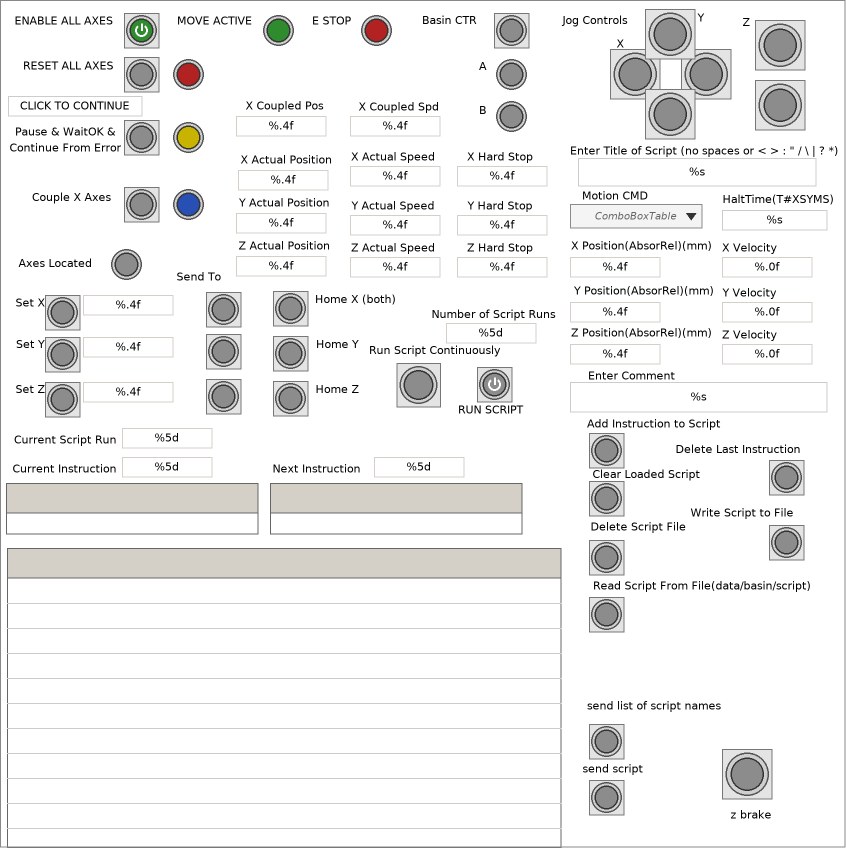
VISUALIZATION visMotorControl  // 846x848
    Label (12,58 113x16), "RESET ALL AXES"
    Label (12,126 107x12), "Pause & WaitOK &"
    Label (9,13 110x16), "ENABLE ALL AXES"
    Textfield (722,257 90x20), "%.0f", text variable: GVL_MOTION.InstructionBuffer.SetXVelocity
        OnMouseClick: write the text variable via InputWithLimits, min 1, max 300, title 'Enter Speed'
    Textfield (570,257 90x20), "%.4f", text variable: GVL_MOTION.InstructionBuffer.SetXPosition
        OnMouseClick: write the text variable via Default, min -200, max 1500
    Label (722,241 55x14), "X Velocity"
    Label (570,238 143x16), "X Position(AbsorRel)(mm)"
    Label (350,149 86x16), "X Actual Speed"
    Label (238,149 97x22), "X Actual Position"
    Textfield (350,166 90x20), "%.4f", text variable: GVL_MOTION.STATUS.xVelOut
    Textfield (238,170 90x20), "%.4f", text variable: GVL_MOTION.STATUS.xPosOut
    ComboBoxTable (570,204 132x24), variable: GVL_MOTION.InstructionBuffer.MotionCommand, data array: GVL_MOTION.xyzCMDSelect
        p1014161805: 4 - 0 + INT#1
        p3854506369: GVL_MOTION.xyzCMDSelect[INDEX]
    Label (564,185 102x22), "Motion CMD"
    PushSwitch (589,433 35x35), variable: GVL_MOTION.EXT_CTR.CMDADD, behaviour: TAP, style: Switch-PushSwitch-Gray
    Label (588,416 132x16), "Add Instruction to Script"
    PushSwitch (589,481 35x35), variable: GVL_MOTION.EXT_CTR.CMDCLR, behaviour: TOGGLE, style: Switch-PushSwitch-Gray
    Label (588,465 117x19), "Clear Loaded Script"
    Label (445,402 91x16), "RUN SCRIPT"
    PowerSwitch (477,367 35x35), variable: GVL_MOTION.EXT_CTR.CMDRUN, behaviour: TOGGLE, style: Switch-PowerSwitch-Gray
    Label (722,192 113x15), "HaltTime(T#XSYMS)"
    Textfield (722,210 105x20), "%s", text variable: GVL_MOTION.InstructionBuffer.pausetime
        OnMouseClick: write the text variable via Default, min 0, max 2000
    Label (554,12 82x17), "Jog Controls"
    PushSwitch (610,49 50x50), variable: GVL_MOTION.xJogBW, behaviour: TAP, style: Switch-PushSwitch-Gray
    PushSwitch (681,49 50x50), variable: GVL_MOTION.xJogFW, behaviour: TAP, style: Switch-PushSwitch-Gray
    Textfield (8,96 134x20), "CLICK TO CONTINUE", invisible if: GVL_MOTION.TxtBxWaitOK
    Lamp1 (171,57 35x35), variable: GVL_MOTION.STATUS.PowerError, style: Lamp-Lamp1-Red
    PushSwitch (45,295 35x35), variable: GVL_MOTION.EXT_CTR.SETXPOS, behaviour: TAP, style: Switch-PushSwitch-Gray
    PushSwitch (273,291 35x35), variable: GVL_MOTION.EXT_CTR.CMDHOMEX, behaviour: TAP, style: Switch-PushSwitch-Gray
    Label (14,295 33x16), "Set X"
    Label (313,291 85x17), "Home X (both)"
    Textfield (570,302 90x20), "%.4f", text variable: GVL_MOTION.InstructionBuffer.SetYPosition
        OnMouseClick: write the text variable via Default, min -200, max 1500
    Label (570,283 148x16), "Y Position(AbsorRel)(mm)"
    Textfield (722,302 90x20), "%.0f", text variable: GVL_MOTION.InstructionBuffer.SetYVelocity
        OnMouseClick: write the text variable via InputWithLimits, min 1, max 300, title 'Enter Speed'
    Label (722,286 55x14), "Y Velocity"
    Label (350,198 86x16), "Y Actual Speed"
    Label (236,192 97x22), "Y Actual Position"
    Textfield (350,215 90x20), "%.4f", text variable: GVL_MOTION.STATUS.yVelOut
    Textfield (236,213 90x20), "%.4f", text variable: GVL_MOTION.STATUS.yPosOut
    PushSwitch (45,337 35x35), variable: GVL_MOTION.EXT_CTR.SETYPOS, behaviour: TAP, style: Switch-PushSwitch-Gray
    Label (14,337 33x15), "Set Y"
    PushSwitch (645,9 50x50), variable: GVL_MOTION.yJogFW, behaviour: TAP, style: Switch-PushSwitch-Gray
    PushSwitch (645,89 50x50), variable: GVL_MOTION.yJogBW, behaviour: TAP, style: Switch-PushSwitch-Gray
    Label (6,141 119x14), "Continue From Error"
    Lamp1 (359,13 35x35), variable: GVL_MOTION.STATUS.eStop, style: Lamp-Lamp1-Red
    Label (300,13 63x16), "E STOP"
    PushSwitch (124,187 35x35), variable: GVL_MOTION.EXT_CTR.CMDCOUPLE, behaviour: TAP, style: Switch-PushSwitch-Gray
    Label (29,192 85x11), "Couple X Axes"
    Lamp1 (171,187 35x35), variable: GVL_MOTION.STATUS.xCoupled, style: Lamp-Lamp1-Blue
    Label (350,99 98x16), "X Coupled Spd"
    Label (236,95 97x22), "X Coupled Pos"
    Textfield (350,116 90x20), "%.4f", text variable: GVL_MOTION.xCOut.VelocityOut
    Textfield (236,116 90x20), "%.4f", text variable: GVL_MOTION.xCOut.PositionOut
    Label (693,9 16x18), "Y"
    Label (603,29 35x30), "X"
    PushSwitch (755,80 50x50), variable: GVL_MOTION.zJogBW, behaviour: TAP, style: Switch-PushSwitch-Gray
    PushSwitch (755,20 50x50), variable: GVL_MOTION.zJogFW, behaviour: TAP, style: Switch-PushSwitch-Gray
    Label (737,13 19x19), "Z"
    Label (350,240 86x16), "Z Actual Speed"
    Label (236,235 97x22), "Z Actual Position"
    Textfield (350,257 90x20), "%.4f", text variable: GVL_MOTION.STATUS.zVelOut
    Textfield (236,256 90x20), "%.4f", text variable: GVL_MOTION.STATUS.zPosOut
    Textfield (446,323 90x20), "%5d", text variable: GVL_MOTION.EXT_CTR.SCRIPTITERATIONS
        OnMouseClick: write the text variable via Default, min 1, title 'Enter Speed'
    Label (428,307 131x15), "Number of Script Runs"
    Label (12,255 87x17), "Axes Located"
    Table (6,483 252x51), data array: GVL_MOTION.Script[GVL_MOTION.CurInstruction]
        p3854506369: GVL_MOTION.Script[GVL_MOTION.CurInstruction].MotionCommand
        p1892666644: GVL_MOTION.Script[GVL_MOTION.CurInstruction].SetXPosition
        p338671338: GVL_MOTION.Script[GVL_MOTION.CurInstruction].SetXVelocity
        p2170511999: GVL_MOTION.Script[GVL_MOTION.CurInstruction].SetXAccel
        p3723444502: GVL_MOTION.Script[GVL_MOTION.CurInstruction].SetYPosition
        p1218418051: GVL_MOTION.Script[GVL_MOTION.CurInstruction].SetYVelocity
        p746581629: GVL_MOTION.Script[GVL_MOTION.CurInstruction].SetYAccel
        p3104783080: GVL_MOTION.Script[GVL_MOTION.CurInstruction].SetZPosition
        p2501879983: GVL_MOTION.Script[GVL_MOTION.CurInstruction].SetZVelocity
        p7306298: GVL_MOTION.Script[GVL_MOTION.CurInstruction].PauseTime
        p1933151965: GVL_MOTION.Script[GVL_MOTION.CurInstruction].Comment
        p511219082: xPos
        p1755163831: xVel
        p2237128397: yPos
        p505689113: yVel
        p4088588272: zPos
        p2243050616: zVel
    Label (368,343 134x15), "Run Script Continuously"
    PushSwitchLed (396,363 45x44), variable: GVL_MOTION.CMDLOOP_INT, behaviour: TOGGLE, style: Switch-PushSwitchLed-Gray
    Label (12,461 105x16), "Current Instruction"
    Textfield (122,457 90x20), "%5d", text variable: GVL_MOTION.CurInstruction
        OnMouseClick: write the text variable via Default
    Table (270,483 252x51), data array: GVL_MOTION.Script[GVL_MOTION.NextInstruction]
        p3854506369: GVL_MOTION.Script[GVL_MOTION.NextInstruction].MotionCommand
        p1892666644: GVL_MOTION.Script[GVL_MOTION.NextInstruction].SetXPosition
        p338671338: GVL_MOTION.Script[GVL_MOTION.NextInstruction].SetXVelocity
        p2170511999: GVL_MOTION.Script[GVL_MOTION.NextInstruction].SetXAccel
        p3723444502: GVL_MOTION.Script[GVL_MOTION.NextInstruction].SetYPosition
        p1218418051: GVL_MOTION.Script[GVL_MOTION.NextInstruction].SetYVelocity
        p746581629: GVL_MOTION.Script[GVL_MOTION.NextInstruction].SetYAccel
        p3104783080: GVL_MOTION.Script[GVL_MOTION.NextInstruction].SetZPosition
        p2501879983: GVL_MOTION.Script[GVL_MOTION.NextInstruction].SetZVelocity
        p7306298: GVL_MOTION.Script[GVL_MOTION.NextInstruction].PauseTime
        p1933151965: GVL_MOTION.Script[GVL_MOTION.NextInstruction].Comment
        p511219082: xPos
        p2237128397: yPos
        p4088588272: zPos
    Label (264,461 105x16), "Next Instruction"
    Textfield (374,457 90x20), "%5d", text variable: GVL_MOTION.NextInstruction
        OnMouseClick: write the text variable via Default
    Textfield (578,158 238x28), "%s", text variable: GVL_MOTION.EXT_CTR.SCRIPTNAME
        OnMouseClick: write GVL_MOTION.EXT_CTR.SCRIPTNAME via Edit
    Label (563,145 283x12), "Enter Title of Script (no spaces or < > : " / \ | ? *)"
    Lamp1 (109,247 35x35), variable: GVL_MOTION.STATUS.AxesLocated, style: Lamp-Lamp1-Gray
    Label (169,13 91x16), "MOVE ACTIVE"
    Textfield (570,344 90x20), "%.4f", text variable: GVL_MOTION.InstructionBuffer.SetZPosition
        OnMouseClick: write the text variable via Default, min -200, max 1500
    Label (570,325 143x16), "Z Position(AbsorRel)(mm)"
    Textfield (722,344 90x20), "%.0f", text variable: GVL_MOTION.InstructionBuffer.SetZVelocity
        OnMouseClick: write the text variable via InputWithLimits, min 1, max 20, title 'Enter Speed'
    Label (722,328 55x14), "Z Velocity"
    Lamp1 (261,13 35x35), variable: GVL_MOTION.STATUS.MoveActive, style: Lamp-Lamp1-Green
    PowerSwitch (124,13 35x35), variable: GVL_MOTION.AXESEN_INT, behaviour: TOGGLE, style: Switch-PowerSwitch-Green
    PushSwitch (124,120 35x35), variable: GVL_MOTION.EXT_CTR.STOP, behaviour: TAP, style: Switch-PushSwitch-Gray
    PushSwitch (124,57 35x35), variable: GVL_MOTION.EXT_CTR.AxesReset, behaviour: TAP, style: Switch-PushSwitch-Gray
    Lamp1 (171,120 35x35), variable: GVL_MOTION.STATUS.STOP_INT, style: Lamp-Lamp1-Yellow
    Label (13,432 105x16), "Current Script Run"
    Textfield (122,428 90x20), "%5d", text variable: GVL_MOTION.RUN_INDEX
        OnMouseClick: write the text variable via Default
    Table (7,548 554x300), data array: GVL_MOTION.Script
        p1014161805: 99 - 0 + INT#1
        p3854506369: GVL_MOTION.Script[INDEX].MotionCommand
        p1892666644: GVL_MOTION.Script[INDEX].SetXPosition
        p338671338: GVL_MOTION.Script[INDEX].SetXVelocity
        p2170511999: GVL_MOTION.Script[INDEX].SetXAccel
        p3723444502: GVL_MOTION.Script[INDEX].SetYPosition
        p1218418051: GVL_MOTION.Script[INDEX].SetYVelocity
        p746581629: GVL_MOTION.Script[INDEX].SetYAccel
        p3104783080: GVL_MOTION.Script[INDEX].SetZPosition
        p2501879983: GVL_MOTION.Script[INDEX].SetZVelocity
        p7306298: GVL_MOTION.Script[INDEX].PauseTime
        p1933151965: GVL_MOTION.Script[INDEX].Comment
        p511219082: xPos
        p1755163831: xVel
        p2237128397: yPos
        p505689113: yVel
        p4088588272: zPos
        p2243050616: zVel
    Textfield (570,382 257x30), "%s", text variable: GVL_MOTION.InstructionBuffer.Comment
        OnMouseClick: write the text variable via Edit
    Label (571,370 121x12), "Enter Comment"
    PushSwitch (769,460 35x35), variable: GVL_MOTION.EXT_CTR.CMDDEL, behaviour: TOGGLE, style: Switch-PushSwitch-Gray
    Label (671,440 134x19), "Delete Last Instruction"
    PushSwitch (769,525 35x35), variable: GVL_MOTION.EXT_CTR.CMDSCRIPTWRITE, behaviour: TOGGLE, style: Switch-PushSwitch-Gray
    Label (691,505 102x16), "Write Script to File"
    PushSwitch (589,597 35x35), variable: GVL_MOTION.EXT_CTR.CMDSCRIPTREAD, behaviour: TOGGLE, style: Switch-PushSwitch-Gray
    Label (588,578 228x16), "Read Script From File(data/basin/script)"
    PushSwitch (494,13 35x35), variable: GVL_MOTION.EXT_CTR.BASINCTR, behaviour: TAP, style: Switch-PushSwitch-Gray
    Label (415,13 69x15), "Basin CTR"
    PushSwitch (45,382 35x35), variable: GVL_MOTION.EXT_CTR.SETZPOS, behaviour: TAP, style: Switch-PushSwitch-Gray
    Label (14,382 33x15), "Set Z"
    Textfield (83,295 90x20), "%.4f", text variable: GVL_MOTION.EXT_CTR.POSX
        OnMouseClick: write the text variable via Default, min -200, max 1500
    Textfield (83,337 90x20), "%.4f", text variable: GVL_MOTION.EXT_CTR.POSY
        OnMouseClick: write the text variable via Default, min -200, max 1500
    Textfield (83,382 90x20), "%.4f", text variable: GVL_MOTION.EXT_CTR.POSZ
        OnMouseClick: write the text variable via Default, min -200, max 1500
    PushSwitch (273,336 35x35), variable: GVL_MOTION.EXT_CTR.CMDHOMEY, behaviour: TAP, style: Switch-PushSwitch-Gray
    Label (313,336 49x17), "Home Y"
    PushSwitch (273,381 35x35), variable: GVL_MOTION.EXT_CTR.CMDHOMEZ, behaviour: TAP, style: Switch-PushSwitch-Gray
    Label (313,381 49x17), "Home Z"
    Label (457,149 86x16), "X Hard Stop"
    Textfield (457,166 90x20), "%.4f", text variable: GVL_MOTION.STATUS.HardStopLocations[0]
    Label (457,198 86x16), "Y Hard Stop"
    Textfield (457,215 90x20), "%.4f", text variable: GVL_MOTION.STATUS.HardStopLocations[1]
    Label (457,240 86x16), "Z Hard Stop"
    Textfield (457,257 90x20), "%.4f", text variable: GVL_MOTION.STATUS.HardStopLocations[2]
    Lamp1 (494,57 35x35), variable: GVL_MOTION.BASINLAMPA, style: Lamp-Lamp1-Gray
    Lamp1 (494,99 35x35), variable: GVL_MOTION.BASINLAMPB, style: Lamp-Lamp1-Gray
    Label (469,59 28x15), "A"
    Label (469,103 28x15), "B"
    PushSwitch (589,724 35x35), variable: GVL_MOTION.EXT_CTR.CMDREQLIST, behaviour: TOGGLE, style: Switch-PushSwitch-Gray
    Label (584,698 140x16), "send list of script names"
    PushSwitch (589,780 35x35), variable: GVL_MOTION.EXT_CTR.CMDREQSCRIPT, behaviour: TOGGLE, style: Switch-PushSwitch-Gray
    Label (578,761 70x16), "send script"
    PushSwitch (589,540 35x35), variable: GVL_MOTION.EXT_CTR.CMDSCRIPTDEL, behaviour: TOGGLE, style: Switch-PushSwitch-Gray
    Label (592,519 93x16), "Delete Script File"
    PushSwitch (722,749 50x50), variable: GVL_MOTION.ED2008O.ED2008_Output.MDP5001_200_DO_Channel_7_Output, behaviour: TOGGLE, style: Switch-PushSwitch-Gray
    Label (722,809 58x12), "z brake"
    PushSwitch (206,292 35x35), variable: GVL_MOTION.EXT_CTR.MOVEX, behaviour: TAP, style: Switch-PushSwitch-Gray
    PushSwitch (206,334 35x35), variable: GVL_MOTION.EXT_CTR.MOVEY, behaviour: TAP, style: Switch-PushSwitch-Gray
    PushSwitch (206,379 35x35), variable: GVL_MOTION.EXT_CTR.MOVEZ, behaviour: TAP, style: Switch-PushSwitch-Gray
    Label (174,269 50x16), "Send To"
END_VISUALIZATION

(* stored: Version 1.1.0.1, ProductVersion 3.1.4026.18
   Visu visMotorControl: Id {597b15b9-8242-4835-b47f-ab7cbb2aa3c0} *)
